// TIA Portal V18 export
TYPE "UDT_RTDbasic"
// stored: IsFailsafeCompliant false
   STRUCT
      iID : DInt;   // AIs ID for monitoring
      rValue : Real;   // Real value
      iFilterSet : Int;   // Filter value
      rCalibration : Real;   // Scale Min
      rDiv : Real := 100.0;   // Scale Max
      wMark : String["IOmark_string_length"];   // AIs label for monitoring
   END_STRUCT;
END_TYPE
